// TIA Portal V19 export
DATA_BLOCK "FmControl_DB"   // DB26
// stored: InstanceOfName FmControl, InstanceOfType FB
"FmControl"
   // VAR_INPUT
   //    Totalise : Bool;
   //    "Stop & Reset Count" : Bool;
   //    "Stop & Preset Value" : Bool;
   //    "reset and totalise" : Bool;
   //    "Reset  & Restart" : Bool;
   //    "Preset and Start" : Bool;
   //    Hold : Bool;
   // END_VAR
   // VAR_OUTPUT
   //    FmTotaliserControl : Byte;
   // END_VAR
BEGIN
END_DATA_BLOCK
